ABB RobotStudio station: Aristides - Copy_20220201-182259.rsstn

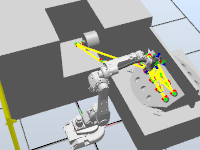
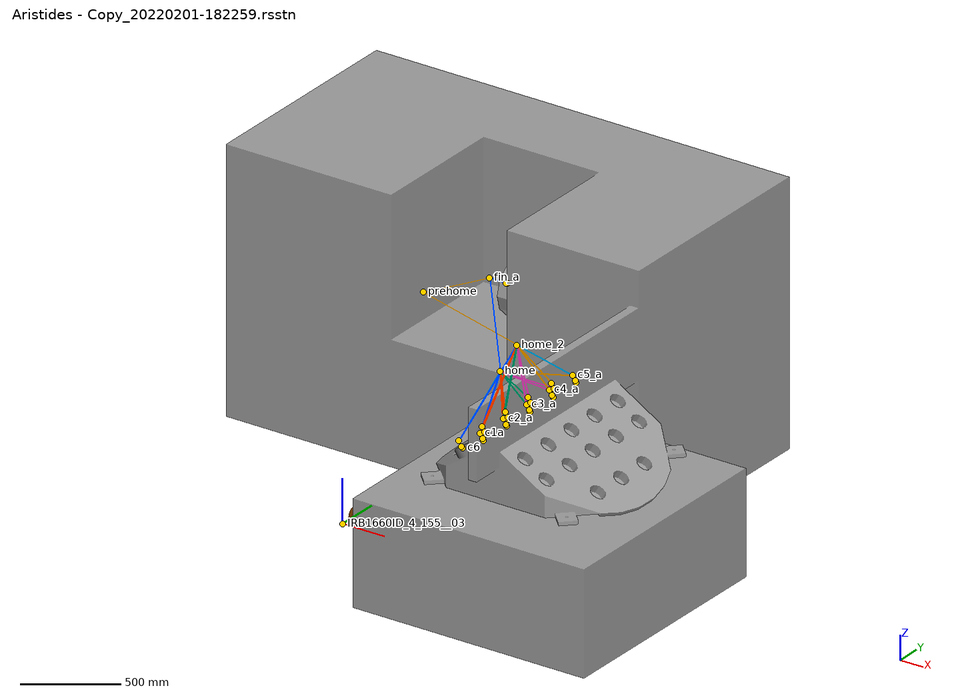
[picture v1: parts stored in the station drawn from their meshes, with robot base, taught points and paths (robot models come from the ABB library and are not in the file)]
Station Station (saved by RobotStudio 21.4.9700.0)
Controller Controller3
  mechanical unit ROB_1: IRB1660ID_4_155__03, 6 joints, base frame (0, 0, 0) mm
Layout (positions relative to the parent item):
  - IRB1660ID_4_155__03 [mechanism, from Robots\IRB1660ID_4_155__03.rslib] at (0, 0, 0) mm; joint values [0, 0.0381, -0.0902, 0, 0.5757, 0] (rad or m)
  - Pinza_1 [mechanism, from Efectores_finales - Copy\Pinza_1.rslib] at (964.87, 0, 1263.64) mm, rotated rx -180 ry 60 rz -180 deg; joint values [0, 0] (rad or m)
  - Conjunto_para_piezas_huecos [part] at (1981.81, -744.19, 0) mm, rotated rx 90 ry 0 rz 180 deg, size 1400 x 1300 x 1400 mm
  - Torno [part] at (-1172.42, 1966.27, 0) mm, rotated rx 0 ry 0 rz 180 deg, size 2500 x 1300 x 1500 mm
  - Fence_740 [graphiccomponentgroup, from Equipment\Fence_740.rslib] at (-1160.76, -802.49, 0) mm
    - Body 1 [part, from Equipment\Fence_740.rslib]
    - Body 2 [part, from Equipment\Fence_740.rslib]
  - Fence_2500 [graphiccomponentgroup, from Equipment\Fence_2500.rslib] at (1297.15, -826.85, 0) mm, rotated rx 0 ry 0 rz 90 deg
    - Body 1 [part, from Equipment\Fence_2500.rslib]
    - Body 2 [part, from Equipment\Fence_2500.rslib]
  - Fence_740_2 [graphiccomponentgroup, from Equipment\Fence_740.rslib] at (-1148.66, -57.63, 0) mm
    - Body 1 [part, from Equipment\Fence_740.rslib]
    - Body 2 [part, from Equipment\Fence_740.rslib]
  - c5 [part] at (1213.21, 355.81, 885.53) mm, rotated rx 0 ry -32 rz 0 deg, size 80 x 79.4 x 100 mm
  - c3 [part] at (1213.21, -44.2, 885.53) mm, rotated rx 0 ry -32 rz 0 deg, size 80 x 79.4 x 100 mm
  - c2 [part] at (1213.21, -244.19, 885.53) mm, rotated rx 0 ry -32 rz 0 deg, size 80 x 79.4 x 100 mm
  - c8 [part] at (1084.59, -44.2, 808.36) mm, rotated rx 0 ry -32 rz 0 deg, size 80 x 79.4 x 100 mm
  - c4 [part] at (1213.21, 155.81, 885.53) mm, rotated rx 0 ry -32 rz 0 deg, size 80 x 79.4 x 100 mm
  - c7 [part] at (1084.59, -244.19, 808.36) mm, rotated rx 0 ry -32 rz 0 deg, size 80 x 79.4 x 100 mm
  - c6 [part] at (1084.59, -444.19, 808.36) mm, rotated rx 0 ry -32 rz 0 deg, size 80 x 79.4 x 100 mm
  - c9 [part] at (1084.59, 155.81, 808.36) mm, rotated rx 0 ry -32 rz 0 deg, size 80 x 79.4 x 100 mm
  - c10 [part] at (1084.59, 355.81, 808.36) mm, rotated rx 0 ry -32 rz 0 deg, size 80 x 79.4 x 100 mm
  - fin [part] at (377.58, 1016.27, 1000) mm, size 100 x 79.4 x 80 mm
  - c0 [part] at (277.58, 1016.27, 1000) mm, size 100 x 79.4 x 80 mm
  - Efector final 2 [part] at (70, 0, -80) mm, rotated rx 0 ry -90 rz -180 deg, size 100 x 99.5 x 30 mm
  - Pinza1_5 [part] at (130, 10, -10) mm, rotated rx 0 ry 0 rz 180 deg, size 60 x 20 x 60 mm
  - Pinza1_6 [part] at (130, -10, 150) mm, rotated rx 180 ry 0 rz 180 deg, size 60 x 20 x 60 mm
    - Pinza_2_1 [frame] at (30, 10, 80) mm, rotated rx 0 ry -90 rz 0 deg
  - Pinza_2 [mechanism, from Efectores_finales\PINZA2.rslib] at (964.87, 0, 1263.64) mm, rotated rx -180 ry 60 rz -180 deg; joint values [0, 0] (rad or m)
  - CollisionSensor [smart component, from Components\CollisionSensor.rslib]
      properties: Object1=Pinza_2; Object2=(none); NearMiss=0.0001; Part1=(none); Part2=(none); CollisionType=0
  - CollisionSensor_2 [smart component, from Components\CollisionSensor.rslib]
      properties: Object1=Pinza_2; Object2=c0_invisible; NearMiss=0.01; Part1=Torno; Part2=c0; CollisionType=2
  - Attacher [smart component, from Components\Attacher.rslib]
      properties: Parent=Pinza_2; Flange=0; Child=(none); Mount=false; Offset=[0 0 0]; Orientation=[0 0 0]
  - Detacher [smart component, from Components\Detacher.rslib]
      properties: Child=(none); KeepPosition=true
  - CollisionSensor_3 [smart component, from Components\CollisionSensor.rslib]
      properties: Object1=Pinza_1; Object2=c0; NearMiss=0.01; Part1=(none); Part2=(none); CollisionType=0
  - Attacher_2 [smart component, from Components\Attacher.rslib]
      properties: Parent=Pinza_1; Flange=0; Child=(none); Mount=false; Offset=[0 0 0]; Orientation=[0 0 0]
  - Detacher_2 [smart component, from Components\Detacher.rslib]
      properties: Child=(none); KeepPosition=true
  - c1 [part] at (1213.21, -444.19, 885.53) mm, rotated rx 0 ry -32 rz 0 deg, size 80 x 79.4 x 100 mm
  - c0_invisible [part] at (277.58, 1016.27, 1000) mm, size 100 x 79.4 x 80 mm
Attachment: Pinza_2 is attached to IRB1660ID_4_155__03 / Link6
Attachment: Pinza_1 is attached to IRB1660ID_4_155__03 / Link6
Station signals: DO s
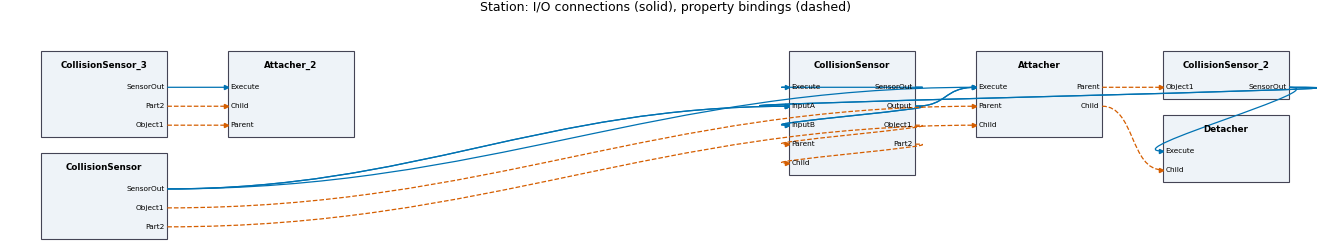
Station logic (signal -> signal, property => property):
  CollisionSensor.SensorOut -> Attacher.Execute
  CollisionSensor_3.SensorOut -> Attacher_2.Execute
  LogicGate_2.Output -> Attacher.Execute
  CollisionSensor_2.SensorOut -> LogicGate.InputA
  LogicGate.Output -> LogicGate_2.InputB
  CollisionSensor.SensorOut -> LogicGate_2.InputA
  CollisionSensor.SensorOut -> LogicGate_4.InputA
  CollisionSensor_2.SensorOut -> LogicGate_3.InputA
  LogicGate_3.Output -> LogicGate_4.InputB
  LogicGate_4.Output -> Attacher.Execute
  CollisionSensor_2.SensorOut -> Detacher.Execute
  CollisionSensor.SensorOut -> Attacher.Execute
  CollisionSensor.Object1 => Attacher.Parent
  CollisionSensor.Part2 => Attacher.Child
  CollisionSensor.Object1 => Attacher.Parent
  CollisionSensor.Part2 => Attacher.Child
  CollisionSensor_3.Part2 => Attacher_2.Child
  CollisionSensor_3.Object1 => Attacher_2.Parent
  Attacher.Parent => CollisionSensor_2.Object1
  Attacher.Child => Detacher.Child
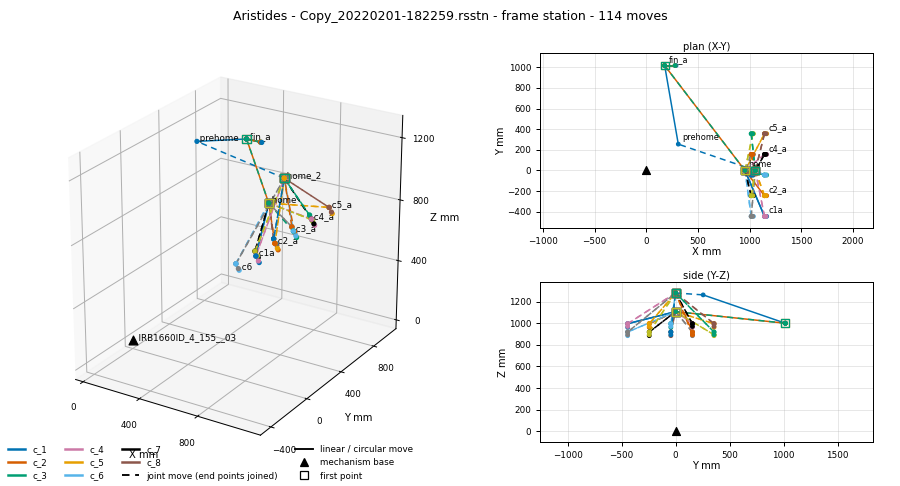
[picture p0: tool path of Aristides - Copy_20220201-182259.rsstn in frame station, 114 of 114 moves have a stored position in this frame; points joined in program order, loops and branches not executed]
Targets, tools, work objects and paths stored in the station, written as RAPID:
! task T_ROB1
MODULE Module1
  CONST robtarget home:=[[955.495207776,0,1107.397459622],[0.258819045,0,-0.965925826,0],[0,0,0,0],[9E+09,9E+09,9E+09,9E+09,9E+09,9E+09]];
  CONST robtarget c1:=[[1165.520192645,-444.195,961.85451904],[0.275637356,0,0.961261696,0],[-1,1,-2,0],[9E+09,9E+09,9E+09,9E+09,9E+09,9E+09]];
  CONST robtarget c1a:=[[1144.323422065,-444.195,995.77644288],[0.275637356,0,0.961261696,0],[-1,1,-2,0],[9E+09,9E+09,9E+09,9E+09,9E+09,9E+09]];
  CONST robtarget c2:=[[1165.520192645,-244.195,961.85451904],[0.275637356,0,0.961261696,0],[-1,1,-2,0],[9E+09,9E+09,9E+09,9E+09,9E+09,9E+09]];
  CONST robtarget c2_a:=[[1144.323422065,-244.195,995.77644288],[0.275637356,0,0.961261696,0],[-1,1,-2,0],[9E+09,9E+09,9E+09,9E+09,9E+09,9E+09]];
  CONST robtarget c3:=[[1165.520192645,-44.195,961.85451904],[0.275637356,0,0.961261696,0],[-1,-1,0,1],[9E+09,9E+09,9E+09,9E+09,9E+09,9E+09]];
  CONST robtarget c3_a:=[[1144.323422065,-44.195,995.77644288],[0.275637356,0,0.961261696,0],[-1,-1,0,1],[9E+09,9E+09,9E+09,9E+09,9E+09,9E+09]];
  CONST robtarget c4:=[[1165.520192645,155.805,961.85451904],[0.275637356,0,0.961261696,0],[0,-2,1,0],[9E+09,9E+09,9E+09,9E+09,9E+09,9E+09]];
  CONST robtarget c4_a:=[[1144.323422065,155.805,995.77644288],[0.275637356,0,0.961261696,0],[0,-2,1,0],[9E+09,9E+09,9E+09,9E+09,9E+09,9E+09]];
  CONST robtarget c5:=[[1165.520192645,355.805,961.85451904],[0.275637356,0,0.961261696,0],[0,-2,1,0],[9E+09,9E+09,9E+09,9E+09,9E+09,9E+09]];
  CONST robtarget c5_a:=[[1144.323422065,355.805,995.77644288],[0.275637356,0,0.961261696,0],[0,-2,1,0],[9E+09,9E+09,9E+09,9E+09,9E+09,9E+09]];
  CONST robtarget c6:=[[1036.896192645,-444.195,884.68051904],[0.275637356,0,0.961261696,0],[-1,1,-2,0],[9E+09,9E+09,9E+09,9E+09,9E+09,9E+09]];
  CONST robtarget c6_a:=[[1015.699422065,-444.195,918.60244288],[0.275637356,0,0.961261696,0],[-1,1,-2,0],[9E+09,9E+09,9E+09,9E+09,9E+09,9E+09]];
  CONST robtarget c7:=[[1036.896192645,-244.195,884.68051904],[0.275637356,0,0.961261696,0],[-1,1,-2,0],[9E+09,9E+09,9E+09,9E+09,9E+09,9E+09]];
  CONST robtarget c7_a:=[[1015.699422065,-244.195,918.60244288],[0.275637356,0,0.961261696,0],[-1,1,-2,0],[9E+09,9E+09,9E+09,9E+09,9E+09,9E+09]];
  CONST robtarget c8:=[[1036.896192645,-44.195,884.68051904],[0.275637356,0,0.961261696,0],[-1,-1,0,1],[9E+09,9E+09,9E+09,9E+09,9E+09,9E+09]];
  CONST robtarget c8_a:=[[1015.699422065,-44.195,918.60244288],[0.275637356,0,0.961261696,0],[-1,-1,0,1],[9E+09,9E+09,9E+09,9E+09,9E+09,9E+09]];
  CONST robtarget c9_a:=[[1015.699422065,155.805,918.60244288],[0.275637356,0,0.961261696,0],[0,-2,1,0],[9E+09,9E+09,9E+09,9E+09,9E+09,9E+09]];
  CONST robtarget c9:=[[1036.896192645,155.805,884.68051904],[0.275637356,0,0.961261696,0],[0,-2,1,0],[9E+09,9E+09,9E+09,9E+09,9E+09,9E+09]];
  CONST robtarget c10:=[[1036.896192645,355.805,884.68051904],[0.275637356,0,0.961261696,0],[0,-2,1,0],[9E+09,9E+09,9E+09,9E+09,9E+09,9E+09]];
  CONST robtarget c10_a:=[[1031.597,355.805,893.161],[0.275637356,0,0.961261696,0],[0,-2,1,0],[9E+09,9E+09,9E+09,9E+09,9E+09,9E+09]];
  CONST robtarget fin_a:=[[177.584,1016.268,1000],[0.5,0.5,0.5,0.5],[0,1,-1,0],[9E+09,9E+09,9E+09,9E+09,9E+09,9E+09]];
  CONST robtarget fin:=[[287.584,1016.268,1000],[0.5,0.5,0.5,0.5],[0,1,-1,0],[9E+09,9E+09,9E+09,9E+09,9E+09,9E+09]];
  CONST robtarget home_2:=[[1055.495207776,0,1280.602540378],[0.965925826,0,0.258819045,0],[0,0,0,0],[9E+09,9E+09,9E+09,9E+09,9E+09,9E+09]];
  CONST robtarget final_a:=[[177.584,1016.268,1000],[0.5,-0.5,0.5,-0.5],[0,0,0,0],[9E+09,9E+09,9E+09,9E+09,9E+09,9E+09]];
  CONST robtarget final:=[[278.084,1016.268,1000],[0.5,-0.5,0.5,-0.5],[0,1,1,0],[9E+09,9E+09,9E+09,9E+09,9E+09,9E+09]];
  CONST robtarget prehome:=[[309.604,254.998,1262.538],[0.396697298,0.585347123,0.410036045,0.576081975],[0,1,0,0],[9E+09,9E+09,9E+09,9E+09,9E+09,9E+09]];
  CONST robtarget c1_3:=[[1160.221,-444.195,970.335],[0,0.961261696,0,0.275637356],[-1,1,0,0],[9E+09,9E+09,9E+09,9E+09,9E+09,9E+09]];
  CONST robtarget c1a_3:=[[1144.323422065,-444.195,995.77644288],[0,0.961261696,0,0.275637356],[-1,1,0,0],[9E+09,9E+09,9E+09,9E+09,9E+09,9E+09]];
  CONST robtarget c2_3:=[[1160.221,-244.195,970.335],[0,0.961261696,0,0.275637356],[-1,1,0,0],[9E+09,9E+09,9E+09,9E+09,9E+09,9E+09]];
  CONST robtarget c2_a_2:=[[1144.323422065,-244.195,995.77644288],[0,0.961261696,0,0.275637356],[-1,1,0,0],[9E+09,9E+09,9E+09,9E+09,9E+09,9E+09]];
  CONST robtarget c3_3:=[[1160.221,-44.195,970.335],[0,0.961261696,0,0.275637356],[-1,-1,-2,1],[9E+09,9E+09,9E+09,9E+09,9E+09,9E+09]];
  CONST robtarget c3_a_2:=[[1144.323422065,-44.195,995.77644288],[0,0.961261696,0,0.275637356],[-1,-1,-2,1],[9E+09,9E+09,9E+09,9E+09,9E+09,9E+09]];
  CONST robtarget c4_3:=[[1160.221,155.805,970.335],[0,0.961261696,0,0.275637356],[0,-2,-1,0],[9E+09,9E+09,9E+09,9E+09,9E+09,9E+09]];
  CONST robtarget c4_a_2:=[[1144.323422065,155.805,995.77644288],[0,0.961261696,0,0.275637356],[0,-2,-1,0],[9E+09,9E+09,9E+09,9E+09,9E+09,9E+09]];
  CONST robtarget c5_3:=[[1160.221,355.805,970.335],[0,0.961261696,0,0.275637356],[0,-2,-1,0],[9E+09,9E+09,9E+09,9E+09,9E+09,9E+09]];
  CONST robtarget c5_a_2:=[[1144.323422065,355.805,995.77644288],[0,0.961261696,0,0.275637356],[0,-2,-1,0],[9E+09,9E+09,9E+09,9E+09,9E+09,9E+09]];
  CONST robtarget c6_3:=[[1031.597,-444.195,893.161],[0,0.961261696,0,0.275637356],[-1,1,0,0],[9E+09,9E+09,9E+09,9E+09,9E+09,9E+09]];
  CONST robtarget c6_a_2:=[[1015.699422065,-444.195,918.60244288],[0,0.961261696,0,0.275637356],[-1,1,0,0],[9E+09,9E+09,9E+09,9E+09,9E+09,9E+09]];
  CONST robtarget c7_3:=[[1031.597,-244.195,893.161],[0,0.961261696,0,0.275637356],[-1,1,0,0],[9E+09,9E+09,9E+09,9E+09,9E+09,9E+09]];
  CONST robtarget c7_a_2:=[[1015.699422065,-244.195,918.60244288],[0,0.961261696,0,0.275637356],[-1,1,0,0],[9E+09,9E+09,9E+09,9E+09,9E+09,9E+09]];
  CONST robtarget c8_3:=[[1031.597,-44.195,893.161],[0,0.961261696,0,0.275637356],[-1,-1,-2,1],[9E+09,9E+09,9E+09,9E+09,9E+09,9E+09]];
  CONST robtarget c8_a_2:=[[1015.699422065,-44.195,918.60244288],[0,0.961261696,0,0.275637356],[-1,-1,-2,1],[9E+09,9E+09,9E+09,9E+09,9E+09,9E+09]];
  CONST robtarget c9_2:=[[1031.597,155.805,893.161],[0,0.961261696,0,0.275637356],[0,-2,-1,0],[9E+09,9E+09,9E+09,9E+09,9E+09,9E+09]];
  CONST robtarget c9_a_3:=[[1015.699422065,155.805,918.60244288],[0,0.961261696,0,0.275637356],[0,-2,-1,0],[9E+09,9E+09,9E+09,9E+09,9E+09,9E+09]];
  CONST robtarget c10_3:=[[1031.597,355.805,893.161],[0,0.961261696,0,0.275637356],[0,-2,-1,0],[9E+09,9E+09,9E+09,9E+09,9E+09,9E+09]];
  CONST robtarget c10_a_2:=[[1015.699422065,355.805,918.60244288],[0,0.961261696,0,0.275637356],[0,-2,-1,0],[9E+09,9E+09,9E+09,9E+09,9E+09,9E+09]];
  PROC main()
    c_1;
    c_1_2;
    c_2;
    c_2_2;
    c_3;
    c_3_2;
    c_4;
    c_4_2;
    c_5;
    c_5_2;
    c_6;
    c_6_2;
    c_7;
    c_7_2;
    c_8;
    c_8_2;
    c_9;
    c_10;
    c_9_2;
    c_10_2;
    giro;
    torno;
  ENDPROC
  PROC c_1()
    MoveJ home,v1000,z100,Pinza_2_1\WObj:=Workobject_2;
    MoveL c1a,v1000,z100,Pinza_2_1\WObj:=Workobject_2;
    MoveL c1,v1000,fine,Pinza_2_1\WObj:=Workobject_2;
    MoveL c1a,v1000,z100,Pinza_2_1\WObj:=Workobject_2;
    MoveL home,v1000,z100,Pinza_2_1\WObj:=Workobject_2;
  ENDPROC
  PROC c_2()
    MoveJ home,v1000,z100,Pinza_2_1\WObj:=Workobject_2;
    MoveJ c2_a,v1000,z100,Pinza_2_1\WObj:=Workobject_2;
    MoveJ c2,v1000,z100,Pinza_2_1\WObj:=Workobject_2;
    MoveJ c2_a,v1000,z100,Pinza_2_1\WObj:=Workobject_2;
    MoveJ home,v1000,z100,Pinza_2_1\WObj:=Workobject_2;
  ENDPROC
  PROC c_3()
    MoveJ home,v1000,z100,Pinza_2_1\WObj:=Workobject_2;
    MoveJ c3_a,v1000,z100,Pinza_2_1\WObj:=Workobject_2;
    MoveJ c3,v1000,z100,Pinza_2_1\WObj:=Workobject_2;
    MoveJ c3_a,v1000,z100,Pinza_2_1\WObj:=Workobject_2;
    MoveJ home,v1000,z100,Pinza_2_1\WObj:=Workobject_2;
  ENDPROC
  PROC c_4()
    MoveJ home,v1000,z100,Pinza_2_1\WObj:=Workobject_2;
    MoveJ c4_a,v1000,z100,Pinza_2_1\WObj:=Workobject_2;
    MoveJ c4,v1000,z100,Pinza_2_1\WObj:=Workobject_2;
    MoveJ c4_a,v1000,z100,Pinza_2_1\WObj:=Workobject_2;
    MoveJ home,v1000,z100,Pinza_2_1\WObj:=Workobject_2;
  ENDPROC
  PROC c_5()
    MoveJ home,v1000,z100,Pinza_2_1\WObj:=Workobject_2;
    MoveJ c5_a,v1000,z100,Pinza_2_1\WObj:=Workobject_2;
    MoveJ c5,v1000,z100,Pinza_2_1\WObj:=Workobject_2;
    MoveJ c5_a,v1000,z100,Pinza_2_1\WObj:=Workobject_2;
    MoveJ home,v1000,z100,Pinza_2_1\WObj:=Workobject_2;
  ENDPROC
  PROC c_6()
    MoveJ home,v1000,z100,Pinza_2_1\WObj:=Workobject_2;
    MoveJ c6_a,v1000,z100,Pinza_2_1\WObj:=Workobject_2;
    MoveJ c6,v1000,z100,Pinza_2_1\WObj:=Workobject_2;
    MoveJ c6_a,v1000,z100,Pinza_2_1\WObj:=Workobject_2;
    MoveJ home,v1000,z100,Pinza_2_1\WObj:=Workobject_2;
  ENDPROC
  PROC c_7()
    MoveJ home,v1000,z100,Pinza_2_1\WObj:=Workobject_2;
    MoveJ c7_a,v1000,z100,Pinza_2_1\WObj:=Workobject_2;
    MoveJ c7,v1000,z100,Pinza_2_1\WObj:=Workobject_2;
    MoveJ c7_a,v1000,z100,Pinza_2_1\WObj:=Workobject_2;
    MoveJ home,v1000,z100,Pinza_2_1\WObj:=Workobject_2;
  ENDPROC
  PROC c_8()
    MoveJ home,v1000,z100,Pinza_2_1\WObj:=Workobject_2;
    MoveJ c8_a,v1000,z100,Pinza_2_1\WObj:=Workobject_2;
    MoveJ c8,v1000,z100,Pinza_2_1\WObj:=Workobject_2;
    MoveJ c8_a,v1000,z100,Pinza_2_1\WObj:=Workobject_2;
    MoveJ home,v1000,z100,Pinza_2_1\WObj:=Workobject_2;
  ENDPROC
  PROC c_9()
    MoveJ home,v1000,z100,Pinza_2_1\WObj:=Workobject_2;
    MoveJ c9_a,v1000,z100,Pinza_2_1\WObj:=Workobject_2;
    MoveJ c9,v1000,z100,Pinza_2_1\WObj:=Workobject_2;
    MoveJ c9_a,v1000,z100,Pinza_2_1\WObj:=Workobject_2;
    MoveJ home,v1000,z100,Pinza_2_1\WObj:=Workobject_2;
  ENDPROC
  PROC c_10()
    MoveJ home,v1000,z100,Pinza_2_1\WObj:=Workobject_2;
    MoveJ c10_a,v1000,z100,Pinza_2_1\WObj:=Workobject_2;
    MoveJ c10,v1000,z100,Pinza_2_1\WObj:=Workobject_2;
    MoveJ c10_a,v1000,z100,Pinza_2_1\WObj:=Workobject_2;
    MoveJ home,v1000,z100,Pinza_2_1\WObj:=Workobject_2;
  ENDPROC
  PROC torno()
    MoveJ home_2,v1000,z100,Pinza_1\WObj:=Workobject_4;
    MoveJ prehome,v1000,z100,Pinza_1\WObj:=Workobject_4;
    MoveL fin_a,v1000,z100,Pinza_1\WObj:=Workobject_4;
    MoveL fin,v1000,z100,Pinza_1\WObj:=Workobject_4;
    MoveL fin_a,v1000,z100,Pinza_1\WObj:=Workobject_4;
  ENDPROC
  PROC giro()
    MoveJ final_a,v1000,z100,Pinza_2_1\WObj:=Workobject_2;
    MoveL final,v1000,fine,Pinza_2_1\WObj:=Workobject_2;
    MoveL final_a,v1000,z100,Pinza_2_1\WObj:=Workobject_2;
    MoveL home,v1000,z100,Pinza_2_1\WObj:=Workobject_2;
  ENDPROC
  PROC Path_10()
    MoveJ final_a,v1000,z100,tool0\WObj:=Workobject_2;
    MoveJ final,v1000,z100,tool0\WObj:=Workobject_2;
    MoveJ final_a,v1000,z100,tool0\WObj:=Workobject_2;
    MoveJ home,v1000,z100,tool0\WObj:=Workobject_2;
  ENDPROC
  PROC c_1_2()
    MoveJ home_2,v1000,z100,Pinza_1\WObj:=Workobject_4;
    MoveJ c1a_3,v1000,z100,Pinza_1\WObj:=Workobject_4;
    MoveJ c1_3,v1000,z100,Pinza_1\WObj:=Workobject_4;
    MoveJ c1a_3,v1000,z100,Pinza_1\WObj:=Workobject_4;
    MoveJ home_2,v1000,z100,Pinza_1\WObj:=Workobject_4;
  ENDPROC
  PROC c_2_2()
    MoveJ home_2,v1000,z100,Pinza_1\WObj:=Workobject_4;
    MoveJ c2_a_2,v1000,z100,Pinza_1\WObj:=Workobject_4;
    MoveJ c2_3,v1000,z100,Pinza_1\WObj:=Workobject_4;
    MoveJ c2_a_2,v1000,z100,Pinza_1\WObj:=Workobject_4;
    MoveJ home_2,v1000,z100,Pinza_1\WObj:=Workobject_4;
  ENDPROC
  PROC c_3_2()
    MoveJ home_2,v1000,z100,Pinza_1\WObj:=Workobject_4;
    MoveJ c3_a_2,v1000,z100,Pinza_1\WObj:=Workobject_4;
    MoveJ c3_3,v1000,z100,Pinza_1\WObj:=Workobject_4;
    MoveJ c3_a_2,v1000,z100,Pinza_1\WObj:=Workobject_4;
    MoveJ home_2,v1000,z100,Pinza_1\WObj:=Workobject_4;
  ENDPROC
  PROC c_4_2()
    MoveJ home_2,v1000,z100,Pinza_1\WObj:=Workobject_4;
    MoveJ c4_a_2,v1000,z100,Pinza_1\WObj:=Workobject_4;
    MoveJ c4_3,v1000,z100,Pinza_1\WObj:=Workobject_4;
    MoveJ c4_a_2,v1000,z100,Pinza_1\WObj:=Workobject_4;
    MoveJ home_2,v1000,z100,Pinza_1\WObj:=Workobject_4;
  ENDPROC
  PROC c_5_2()
    MoveJ home_2,v1000,z100,Pinza_1\WObj:=Workobject_4;
    MoveJ c5_a_2,v1000,z100,Pinza_1\WObj:=Workobject_4;
    MoveJ c5_3,v1000,z100,Pinza_1\WObj:=Workobject_4;
    MoveJ c5_a_2,v1000,z100,Pinza_1\WObj:=Workobject_4;
    MoveJ home_2,v1000,z100,Pinza_1\WObj:=Workobject_4;
  ENDPROC
  PROC c_6_2()
    MoveJ home_2,v1000,z100,Pinza_1\WObj:=Workobject_4;
    MoveJ c6_a_2,v1000,z100,Pinza_1\WObj:=Workobject_4;
    MoveJ c6_3,v1000,z100,Pinza_1\WObj:=Workobject_4;
    MoveJ c6_a_2,v1000,z100,Pinza_1\WObj:=Workobject_4;
    MoveJ home_2,v1000,z100,Pinza_1\WObj:=Workobject_4;
  ENDPROC
  PROC c_7_2()
    MoveJ home_2,v1000,z100,Pinza_1\WObj:=Workobject_4;
    MoveJ c7_a_2,v1000,z100,Pinza_1\WObj:=Workobject_4;
    MoveJ c7_3,v1000,z100,Pinza_1\WObj:=Workobject_4;
    MoveJ c7_a_2,v1000,z100,Pinza_1\WObj:=Workobject_4;
    MoveJ home_2,v1000,z100,Pinza_1\WObj:=Workobject_4;
  ENDPROC
  PROC c_8_2()
    MoveJ home_2,v1000,z100,Pinza_1\WObj:=Workobject_4;
    MoveJ c8_a_2,v1000,z100,Pinza_1\WObj:=Workobject_4;
    MoveJ c8_3,v1000,z100,Pinza_1\WObj:=Workobject_4;
    MoveJ c8_a_2,v1000,z100,Pinza_1\WObj:=Workobject_4;
    MoveJ home_2,v1000,z100,Pinza_1\WObj:=Workobject_4;
  ENDPROC
  PROC c_9_2()
    MoveJ home_2,v1000,z100,Pinza_1\WObj:=Workobject_4;
    MoveJ c9_a_3,v1000,z100,Pinza_1\WObj:=Workobject_4;
    MoveJ c9_2,v1000,z100,Pinza_1\WObj:=Workobject_4;
    MoveJ c9_a_3,v1000,z100,Pinza_1\WObj:=Workobject_4;
    MoveJ c9_2,v1000,z100,Pinza_1\WObj:=Workobject_4;
    MoveJ home_2,v1000,z100,Pinza_1\WObj:=Workobject_4;
  ENDPROC
  PROC c_10_2()
    MoveJ home_2,v1000,z100,Pinza_1\WObj:=Workobject_4;
    MoveJ c10_a_2,v1000,z100,Pinza_1\WObj:=Workobject_4;
    MoveJ c10_3,v1000,z100,Pinza_1\WObj:=Workobject_4;
    MoveJ c10_a_2,v1000,z100,Pinza_1\WObj:=Workobject_4;
    MoveJ home_2,v1000,z100,Pinza_1\WObj:=Workobject_4;
  ENDPROC
ENDMODULE

! task T_ROB1
MODULE CalibData
  TASK PERS wobjdata Workobject_2:=[FALSE,TRUE,"",[[0,0,0],[1,0,0,0]],[[0,0,0],[1,0,0,0]]];
  TASK PERS wobjdata Workobject_4:=[FALSE,TRUE,"",[[0,0,0],[1,0,0,0]],[[0,0,0],[1,0,0,0]]];
  PERS tooldata Pinza_2_1:=[TRUE,[[140,0,70],[0.707106781,0,0.707106781,0]],[1,[0,0,1],[1,0,0,0],0,0,0]];
  PERS tooldata Pinza_1:=[TRUE,[[-100,0,70],[0.707106781,0,-0.707106781,0]],[1,[0,0,1],[1,0,0,0],0,0,0]];
  PERS tooldata Vara:=[TRUE,[[0,0,250],[0.707106781,0,0,0.707106781]],[1,[0,0,1],[1,0,0,0],0,0,0]];
  PERS tooldata Soplador:=[TRUE,[[0,-70,70],[0.5,0.5,-0.5,0.5]],[1,[0,0,1],[1,0,0,0],0,0,0]];
ENDMODULE

